// TIA Portal V16 export
// export: Created 2021-05-25T16:14:39.6168044Z, ExportSetting WithDefaults, DisplayName Totally Integrated Automation Portal, DisplayVersion V16, DisplayName TIA Portal Version Control Interface, DisplayVersion V16, DisplayName TIA Portal Openness, DisplayVersion V16, DisplayName STEP 7 Professional, DisplayVersion V16, DisplayName STEP 7 Safety, DisplayVersion V16, DisplayName WinCC Unified SCADA Engineering System, DisplayVersion V16
DATA_BLOCK "dbDI"   // DB10
{ S7_Optimized_Access := 'FALSE'; DB_Accessible_From_OPC_UA := 'FALSE' }
VERSION : 0.1
// stored: AutoNumber false, DBAccessibleFromOPCUA false, IsOnlyStoredInLoadMemory false, IsWriteProtectedInAS false
   VAR
      ZAUSTAVITEV_V_SILI_NI_AKTIVIRANA : Bool;   // 0=NOT OK, 1=OK
      FOTO_ZAVESA_KANAL_1 : Bool;   // 0=NOT OK, 1=OK
      FOTO_ZAVESA_KANAL_2 : Bool;   // 0=NOT OK, 1=OK
      START_LEVO_NA_VPENJANJU : Bool;
      START_DESNO_NA_VPENJANJU : Bool;
      Spare0_5 : Bool;
      Spare0_6 : Bool;
      PRISOTNOST_ZRAKA_NA_NAPRAVI : Bool;   // 0=NOT OK, 1=OK
      Spare1_0 : Bool;
      Spare1_1 : Bool;
      Spare1_2 : Bool;
      Spare1_3 : Bool;
      Spare1_4 : Bool;
      Spare1_5 : Bool;
      Spare1_6 : Bool;
      Spare1_7 : Bool;
      BIMETAL_TRANSPORTA_NOGIC_IZKLJUCIL : Bool;   // (I0.0) / 0=NOT OK, 1=OK
      VIBRATOR_NOGIC_READY : Bool;   // (I0.1) / 0=NOT READY, 1=READY
      BIMETAL_VIJACENJA_NOGIC_IZKLJUCIL : Bool;   // (I0.2) / 0=NOT OK, 1=OK
      FR_MOTORJA1_ZADAJ_DESNO_READY : Bool;   // (I0.3) / 0=NOT READY, 1=READY
      FR_MOTORJA2_SPREDAJ_DESNO_READY : Bool;   // (I0.4) / 0=NOT READY, 1=READY
      FR_MOTORJA1_ZADAJ_LEVO_READY : Bool;   // (I0.5) / 0=NOT READY, 1=READY
      FR_MOTORJA2_SPREDAJ_LEVO_READY : Bool;   // (I0.6) / 0=NOT READY, 1=READY
      Spare20_7 : Bool;
      FOTOCELICA_TRANSPORTA_NOGIC : Bool;   // (I0.7) / 0=NI PRISOTNO, 1=PRISOTNO | NOT USED
      FOTOCELICA_VSTOP_DRCA_NOGIC : Bool;   // (I1.0) / 0=NI PRISOTNO, 1=PRISOTNO | ? | NOT USED
      FOTOCELICA_PRED_MESTOM_LOCEVANJA : Bool;   // (I1.1) / 0=NI PRISOTNO, 1=PRISOTNO | NOT USED
      FOTOCELICA_VSTOP_DRCA_LEVO : Bool;   // (I1.2) / 0=NI PRISOTNO, 1=PRISOTNO | NOT USED
      FOTOCELICA_VSTOP_DRCA_DESNO : Bool;   // (I1.3) / 0=NI PRISOTNO, 1=PRISOTNO | NOT USED
      FOTOCELICA_LOC_IZH_DRCA_LEVO : Bool;   // (I1.4) / 0=NI PRISOTNO, 1=PRISOTNO | NOT USED
      FOTOCELICA_LOC_IZH_DRCA_DESNO : Bool;   // (I1.5) / 0=NI PRISOTNO, 1=PRISOTNO | NOT USED
      NOGICE_V_VIBRATORJU : Bool;
      ROTACIJSKI_CIL_DESNO : Bool;   // 0=NI PRISOTNO, 1=PRISOTNO
      ROTACIJSKI_CIL_SREDINA : Bool;   // 0=NI PRISOTNO, 1=PRISOTNO
      ROTACIJSKI_CIL_LEVO : Bool;   // 0=NI PRISOTNO, 1=PRISOTNO
      LOC_DRCA_DESNO_NAPREJ : Bool;   // 0=NI PRISOTNO, 1=PRISOTNO | NOT USED
      LOC_DRCA_DESNO_NAZAJ : Bool;   // 0=NI PRISOTNO, 1=PRISOTNO | NOT USED
      LOC_DRCA_LEVO_NAZAJ : Bool;   // 0=NI PRISOTNO, 1=PRISOTNO | NOT USED
      LOC_DRCA_LEVO_NAPREJ : Bool;   // 0=NI PRISOTNO, 1=PRISOTNO | NOT USED
      Spare22_7 : Bool;
      FOTOCELICA_LOC_TRAK_DESNO1 : Bool;   // 0=NI PRISOTNO, 1=PRISOTNO | NOT USED
      FOTOCELICA_LOC_TRAK_DESNO2 : Bool;   // 0=NI PRISOTNO, 1=PRISOTNO | NOT USED
      FOTOCELICA_VIJACENJE_DESNOZADAJ : Bool;   // 0=NI PRISOTNO, 1=PRISOTNO | NOT USED
      FOTOCELICA_VIJACENJE_DESNOSPREDAJ : Bool;   // 0=NI PRISOTNO, 1=PRISOTNO | NOT USED
      VIJACENJE_DESNO_1_NAZAJ : Bool;   // LOCEVANJE NA TRAKU DESNO NAZAJ
      VIJACENJE_DESNO_1_NAPREJ : Bool;   // LOCEVANJE NA TRAKU DESNO NAPREJ
      MESTO_VIJAC_STOP_DESNO_ZAD_NAZAJ : Bool;   // 0=NI PRISOTNO, 1=PRISOTNO
      MESTO_VIJAC_STOP_DESNO_ZAD_NAPREJ : Bool;   // 0=NI PRISOTNO, 1=PRISOTNO
      MESTO_VIJACENJE_DESNO_ZAD_DVIG_DOL : Bool;   // (I1.6) / 0=NI PRISOTNO, 1=PRISOTNO | ? Detekcija spodnje lege cilindra spusta| DONE Man
      MESTO_VIJACENJE_DESNO_ZAD_CENT_NARAZEN : Bool;   // (I1.7) / 0=NI PRISOTNO, 1=PRISOTNO
      MESTO_VIJACENJE_DESNO_ZAD_CENT_SKUPAJ : Bool;   // 0=NI PRISOTNO, 1=PRISOTNO
      Spare24_3 : Bool;   // MESTO_VIJACENJE_DESNO_SPRED_NAZAJ "STOP_DESNO_SPRED_NAZAJ(Spare23_4) ne obstaja. Konec traka ne obstaja cilinder za stopanje nogice.
      Spare24_4 : Bool;   // MESTO_VIJACENJE_DESNO_SPRED_NAPREJ "STOP_DESNO_SPRED_NAPREJ (Spare23_5) ne obstaja. Konec traka ne obstaja cilinder za stopanje nogice.
      MESTO_VIJACENJE_DESNO_SPRED_DVIG_DOL : Bool;   // 0=NI PRISOTNO, 1=PRISOTNO | ? Detekcija spodnje lege cilindra spusta| DONE Man
      MESTO_VIJACENJE_DESNO_SPRED_CENT_NARAZEN : Bool;   // 0=NI PRISOTNO, 1=PRISOTNO
      MESTO_VIJACENJE_DESNO_SPRED_CENT_SKUPAJ : Bool;   // 0=NI PRISOTNO, 1=PRISOTNO
      KONCNA_POZICIJA_VIJACENJA_DES_NAZAJ : Bool;   // 0=NI PRISOTNO, 1=PRISOTNO | NOT USED
      KONCNA_POZICIJA_VIJACENJA_DES_NAPREJ : Bool;   // 0=NI PRISOTNO, 1=PRISOTNO | NOT USED
      Spare25_2 : Bool;
      Spare25_3 : Bool;
      KONCNA_POZICIJA_VIJACENJA_LEVO_NAZAJ : Bool;   // 0=NI PRISOTNO, 1=PRISOTNO | NOT USED
      KONCNA_POZICIJA_VIJACENJA_LEVO_NAPREJ : Bool;   // 0=NI PRISOTNO, 1=PRISOTNO | NOT USED
      Spare25_6 : Bool;
      Spare25_7 : Bool;
      FOTOCELICA_LOC_TRAK_LEVO1 : Bool;   // 0=NI PRISOTNO, 1=PRISOTNO | NOT USED
      FOTOCELICA_LOC_TRAK_LEVO2 : Bool;   // 0=NI PRISOTNO, 1=PRISOTNO | NOT USED
      FOTOCELICA_VIJACENJE_LEVO_ZADAJ : Bool;   // 0=NI PRISOTNO, 1=PRISOTNO | NOT USED
      FOTOCELICA_VIJACENJE_LEVO_SPREDAJ : Bool;   // 0=NI PRISOTNO, 1=PRISOTNO | NOT USED
      VIJACENJE_LEVO_1_NAZAJ : Bool;   // LOCEVANJE NA TRAKU LEVO NAZAJ
      VIJACENJE_LEVO_1_NAPREJ : Bool;   // LOCEVANJE NA TRAKU LEVO NAPREJ
      MESTO_VIJAC_STOP_LEVO_ZAD_NAZAJ : Bool;   // 0=NI PRISOTNO, 1=PRISOTNO
      MESTO_VIJAC_STOP_LEVO_ZAD_NAPREJ : Bool;   // 0=NI PRISOTNO, 1=PRISOTNO
      MESTO_VIJACENJE_LEVO_ZAD_DVIG_DOL : Bool;   // 0=NI PRISOTNO, 1=PRISOTNO | ? Detekcija spodnje lege cilindra spusta| DONE Man
      MESTO_VIJACENJE_LEVO_ZAD_CENT_NARAZEN : Bool;   // 0=NI PRISOTNO, 1=PRISOTNO
      MESTO_VIJACENJE_LEVO_ZAD_CENT_SKUPAJ : Bool;   // 0=NI PRISOTNO, 1=PRISOTNO
      Spare27_3 : Bool;   // MESTO_VIJACENJE_LEVO_SPRED_NAZAJ "STOP_LEVO_SPRED_NAZAJ(Spare26_4) ne obstaja. Konec traka ne obstaja cilinder za stopanje nogice.
      Spare27_4 : Bool;   // MESTO_VIJACENJE_LEVO_SPRED_NAPREJ "STOP_LEVO_SPRED_NAPREJ (Spare26_5) ne obstaja. Konec traka ne obstaja cilinder za stopanje nogice.
      MESTO_VIJACENJE_LEVO_SPRED_DVIG_DOL : Bool;   // 0=NI PRISOTNO, 1=PRISOTNO | ? Detekcija spodnje lege cilindra spusta| DONE Man
      MESTO_VIJACENJE_LEVO_SPRED_CENT_NARAZEN : Bool;   // 0=NI PRISOTNO, 1=PRISOTNO
      MESTO_VIJACENJE_LEVO_SPRED_CENT_SKUPAJ : Bool;   // 0=NI PRISOTNO, 1=PRISOTNO
      INDUKTIVEC_PRAVILNA_VLOZITEV_DNA_1 : Bool;   // 0=NI PRISOTNO, 1=PRISOTNO | NOT USED
      INDUKTIVEC_PRAVILNA_VLOZITEV_DNA_2 : Bool;   // 0=NI PRISOTNO, 1=PRISOTNO | NOT USED
      VPENJANJE_DNA_LEVO_ZADAJ_GOR : Bool;   // 0=NI PRISOTNO, 1=PRISOTNO
      VPENJANJE_DNA_LEVO_ZADAJ_DOL : Bool;   // 0=NI PRISOTNO, 1=PRISOTNO
      VPENJANJE_DNA_LEVO_SPREDAJ_GOR : Bool;   // 0=NI PRISOTNO, 1=PRISOTNO
      VPENJANJE_DNA_LEVO_SPREDAJ_DOL : Bool;   // 0=NI PRISOTNO, 1=PRISOTNO
      VPENJANJE_DNA_DESNO_ZADAJ_GOR : Bool;   // 0=NI PRISOTNO, 1=PRISOTNO
      VPENJANJE_DNA_DESNO_ZADAJ_DOL : Bool;   // 0=NI PRISOTNO, 1=PRISOTNO
      VPENJANJE_DNA_DESNO_SPREDAJ_GOR : Bool;   // 0=NI PRISOTNO, 1=PRISOTNO
      VPENJANJE_DNA_DESNO_SPREDAJ_DOL : Bool;   // 0=NI PRISOTNO, 1=PRISOTNO
      Static_1 : Bool;   // 0=NI PRISOTNO, 1=PRISOTNO
      Spare29_3 : Bool;
      Spare29_4 : Bool;
      Spare29_5 : Bool;
      Spare29_6 : Bool;
      Spare29_7 : Bool;
   END_VAR
BEGIN
END_DATA_BLOCK
